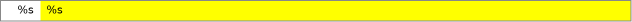
VISUALIZATION V_LoggerMsgLine  // 632x22
VAR_IN_OUT
	IOstLogMsg : ST_LogMessageVisu;
	IOiLogIdAct : INT;
END_VAR
    Rectangle (0,0 40x20)
    Rectangle (30,0 600x20)
    Rectangle (40,0 590x20), colour toggle: IOstLogMsg.iTyp > 1, invisible if: IOstLogMsg.iTyp < 1
    Rectangle (0,0 40x20), "%s", text variable: IOstLogMsg.iLogId, colour toggle: IOstLogMsg.iLogId = IOiLogIdAct, invisible if: IOstLogMsg.iLogId = 0
    Rectangle (40,0 590x20), "%s", text variable: IOstLogMsg.szLogMsg
END_VISUALIZATION

(* stored: Version 1.1.0.1, ProductVersion 3.1.4018.10
   Visu V_LoggerMsgLine: Id {27961802-1c03-496d-9c5c-5940bc967592} *)
